FUNCTION_BLOCK FB_Layer EXTENDS FB_Component IMPLEMENTS I_Layer
VAR_INPUT
END_VAR
VAR_OUTPUT
END_VAR
VAR
	iNext:				I_Component;	// Chain of Responsibility behavioral design pattern 
	fbList:				FB_ListComponent;
END_VAR

METHOD PROTECTED M_Starting : BOOL (* Return state complete*)
VAR
	nIndex: 		DINT;
END_VAR
M_Starting:= TRUE;
WHILE nIndex < fbList.P_Length DO
	IF fbList.M_Index(nIndex).M_RequestState(E_Request.Start) THEN
		;
	ELSE
		M_Starting:= FALSE;
	END_IF	
	nIndex:= nIndex + 1; 
END_WHILE
END_METHOD

{attribute 'OPC.UA.DA.Property' := '1'}
{attribute 'monitoring' := 'call'}
PROPERTY P_List : I_ListComponent
GET
P_List:= fbList;
END_GET
END_PROPERTY

METHOD PROTECTED M_Resetting : BOOL (* Return state complete*)
VAR
	nIndex: 		DINT;
END_VAR
M_Resetting:= TRUE;
WHILE nIndex < fbList.P_Length DO
	IF fbList.M_Index(nIndex).M_RequestState(E_Request.Reset) THEN
		;
	ELSE
		M_Resetting:= FALSE;
	END_IF	
	nIndex:= nIndex + 1; 
END_WHILE
END_METHOD

{attribute 'OPC.UA.DA.Property' := '1'}
{attribute 'monitoring' := 'call'}
PROPERTY PUBLIC P_Next : I_Component
GET
P_Next:= iNext;
END_GET
SET
iNext:= P_Next;
END_SET
END_PROPERTY

METHOD PUBLIC M_Attach
VAR_INPUT
	iComponent:		I_Component;
END_VAR
fbList.M_Add(iComponent);
iComponent.P_Event.P_Observer.M_Attach(THIS^);
fbEvent.P_Observer.M_Attach(iComponent);
END_METHOD

METHOD M_Notify
VAR_INPUT
	stEvent	: ST_Event;
END_VAR
SUPER^.M_Notify(stEvent);
iNext.M_Notify(stEvent);
END_METHOD

METHOD PUBLIC M_Dettach
VAR_INPUT
	iComponent:		I_Component;
END_VAR
fbList.M_Remove(iComponent);
iComponent.P_Event.P_Observer.M_Detach(THIS^);
fbEvent.P_Observer.M_Detach(iComponent);
END_METHOD

END_FUNCTION_BLOCK

(* stored: Version 1.1.0.1
   POU FB_Layer: Id {6c2584ee-5a36-0c50-392e-89c20d77cace}, SpecialFunc None
   Method M_Starting: Id {4e318086-20a9-077e-347c-443a3af7042b}
   Property P_List: Id {5b2e53f7-6521-0d86-3718-b67d38d71e7b}
   Get Get: Id {21be0766-0ebd-0ef1-1a3e-110c16bdb72e}
   Method M_Resetting: Id {6bdcf8ed-efdf-0507-28e5-80bd763eb1d5}
   Property P_Next: Id {bfe686ed-8a9d-0d34-34b1-66bc528ed390}
   Get Get: Id {2f320400-3836-06ec-0636-80ab33c8139d}
   Set Set: Id {9874dbcc-2957-0fba-1736-325d801c41fe}
   Method M_Attach: Id {c25eb90e-66ec-060a-3b43-7637437bb3b8}
   Method M_Notify: Id {debbf766-dd56-0948-0473-018dc5966f2b}
   Method M_Dettach: Id {f13d487a-f32a-0ba9-20c0-98d3bf35cc8f} *)
